FUNCTION A_DWORD : ST_Arg
VAR_INPUT
	nNumber	: REFERENCE TO DWORD;
END_VAR

IF __ISVALIDREF(nNumber) THEN
	A_DWORD.eType := E_ArgType.DWordArg;
	A_DWORD.pData := ADR(nNumber);
	A_DWORD.nSize := SIZEOF(DWORD);
END_IF

END_FUNCTION

(* stored: Version 1.1.0.1, ProductVersion 3.1.4024.15
   POU A_DWORD: Id {83cc648e-b1c2-4629-a03d-6acdef34b847}, SpecialFunc None *)
